FUNCTION_BLOCK FB_Robot_Simulator EXTENDS FB_Robot
VAR_INPUT
    simCellState : eCellState;
    simHydroState : eState;
    HardwareInputs : st_Robot_Input;
END_VAR
VAR_OUTPUT
    HardwareOutputs : st_Robot_Output;
END_VAR
VAR
    simRunningTON : TON := (PT:=T#10S);

    StartupTimeoutTON : TON := (PT:=T#7S);
END_VAR



ExecuteState();
IF NOT (nextState = curState) THEN
	StateTransition();
END_IF;

METHOD abort: BOOL;
VAR_INPUT
END_VAR
IF curState = eState_Running THEN
	nextState := eState_Error;
	abort := TRUE;
ELSE
	abort := FALSE;
END_IF
END_METHOD

ACTION ExecuteState:
// Watch for safety inputs and immediately goto state error
// IF SomeError THEN
//  curState := eState_Error;
// END_IF

CASE curState OF
	eState_Idle: ExecuteState_Idle();
	eState_Startup: ExecuteState_Startup();
	eState_Running: ExecuteState_Running();
    eState_Holding: ExecuteState_Holding();
    eState_Held: ExecuteState_Held();
	eState_Complete: ExecuteState_Complete();
	eState_Error: ExecuteState_Error();
	eState_Independent: ExecuteState_Independent();
END_CASE
END_ACTION

ACTION ExecuteState_Complete:
//Output signals

nextState := eState_Idle;
END_ACTION

ACTION ExecuteState_Error:
//Output signals
HardwareOutputs.fault := TRUE;
END_ACTION

ACTION ExecuteState_Held:
//Set outputs

IF simCellState = eCellState_Error THEN
    // in sim just put it back in idle
    nextState := eState_Idle;
END_IF
END_ACTION

ACTION ExecuteState_Holding:
//Set outputs

//Wait for held signal, then go to Held state
nextState := eState_Held;
END_ACTION

ACTION ExecuteState_Idle:
// monitor IO while idle
// set IO while in idle state

//Output signals
HardwareOutputs.fault := FALSE;
END_ACTION

ACTION ExecuteState_Independent:
//Output signals
END_ACTION

ACTION ExecuteState_Running:


simRunningTON(IN:=TRUE);
IF simRunningTON.Q THEN
    //simRaiseError_counter := simRaiseError_counter+1;
    nextState := eState_Complete;
END_IF

// error robot after nth cycle
//IF simRaiseError_counter = 5 THEN
//    nextState := eState_Error;
//    simRaiseError_counter := 0;
//END_IF
END_ACTION

ACTION ExecuteState_Startup:

nextState := eState_Running;
END_ACTION

METHOD hold : BOOL
IF curState = eState_Running THEN
	nextState := eState_Holding;
	hold := TRUE;
ELSE
	hold := FALSE;
END_IF
END_METHOD

METHOD reset : BOOL
resetAlarms();

IF curState = eState_Complete THEN
	nextState := eState_Idle;
	reset := TRUE;
ELSIF curState = eState_Error THEN // AND InputSignals.AutoMode AND InputSignals.Homed AND InputSignals.LoadUnloadReady AND NOT InputSignals.InCycle THEN
	nextState := eState_Idle;
	reset := TRUE;
ELSE
	reset := FALSE;
END_IF
END_METHOD

METHOD start: BOOL
VAR_INPUT
END_VAR
IF curState = eState_Idle THEN
	nextState := eState_Startup;
	start := TRUE;
ELSE
	start := FALSE;
END_IF
END_METHOD

ACTION StateTransition:
//reset timers watchdog timers

simRunningTON(in := FALSE);
StartupTimeoutTON(IN := FALSE);

IF nextState = eState_Startup THEN
	StartupTimeoutTON(IN := FALSE);
END_IF

IF nextState = eState_Startup THEN
	simRunningTON(IN := FALSE);
END_IF

SUPER^.StateTransition();
END_ACTION

END_FUNCTION_BLOCK

(* stored: Version 1.1.0.1, ProductVersion 3.1.4024.9
   POU FB_Robot_Simulator: Id {8d99ecd9-d781-4c5e-925c-5107575361f0}, SpecialFunc None
   Folder StateMachine: Id {9939dbb8-f0ba-48bc-b044-6d4087b7c50f}
   Folder States: Id {6f0dfb24-3406-4f63-a103-36abc59f6e63}
   Method abort: Id {3edcbad9-26cb-44b3-93f6-d0811cc96895}
   Action ExecuteState: Id {704a6056-e26b-4160-9721-4d4ed178c596}
   Action ExecuteState_Complete: Id {a601be95-9c6d-4835-8e4d-8ffe581055d2}
   Action ExecuteState_Error: Id {8c30d1c0-57f9-4657-a790-5b1d22a55861}
   Action ExecuteState_Held: Id {1c456a31-db40-4a9d-acaa-cbaaba6365f2}
   Action ExecuteState_Holding: Id {b33fd6e1-3976-4583-890e-dc2c14c3e888}
   Action ExecuteState_Idle: Id {66878f2f-6da1-4c50-a6cb-89c19e86c72a}
   Action ExecuteState_Independent: Id {c72d0a9d-15cf-43e7-81bb-5e3a0a9256e9}
   Action ExecuteState_Running: Id {8e637ec5-2ae6-46a6-b16d-91a33e98fe27}
   Action ExecuteState_Startup: Id {f5debea4-afaf-49db-81d0-99c1089f3365}
   Method hold: Id {5ed80ed1-ed16-4b55-abeb-9ec40f1c2cde}
   Method reset: Id {c19f5bf7-8b73-4d49-8310-2acdb4a018f5}
   Method start: Id {4659242a-ad27-4d73-bc37-304f27bf5927}
   Action StateTransition: Id {10ee8015-cceb-4d9b-9037-fc7dafd34547} *)
